(* IEC 61131-3 sources: redes-industriais-mqtt/clp, 4 files *)

(* ---- 1_GVL_MQTT.st ---- *)
(* =========================================================
   GVL_MQTT  -  Global Variable List
   Application > MQTT (pasta) > Add Object > GVL
   ========================================================= *)

VAR_GLOBAL
    (* Estruturas de publicacao e assinatura *)
    Pubs : ARRAY[1..gc_uiMaxPubs] OF MQTT_PUBLISH;
    Subs : ARRAY[1..gc_uiMaxSubs] OF MQTT_SUBSCRIBE;

    (* TOPICOS DE PUBLICACAO - entradas que o CLP envia *)
    PUBLISH_TOPICS : ARRAY[1..gc_uiMaxPubs] OF STRING := [
        'XP340/I_00',
        'XP340/I_01'
    ];

    (* TOPICOS DE ASSINATURA - saidas que o CLP recebe *)
    SUBSCRIBE_TOPICS : ARRAY[1..gc_uiMaxSubs] OF STRING := [
        'XP340/Q_00',
        'XP340/Q_01'
    ];

    (* Status das publicacoes e mensagens recebidas *)
    MQTT_FB_Pub_Status        : ARRAY[1..gc_uiMaxPubs] OF BOOL;
    MQTT_FB_Received_Messages : ARRAY[1..gc_uiMaxSubs] OF MQTT_RECEIVED;

    (* Payloads *)
    PUBS_PAYLOADS : ARRAY[1..gc_uiMaxPubs] OF STRING;
    SUBS_PAYLOADS : ARRAY[1..gc_uiMaxSubs] OF STRING;

    (* Auxiliar - so publica quando o valor muda *)
    PUBS_PAYLOADS_OLD : ARRAY[1..gc_uiMaxPubs] OF STRING;
END_VAR

(* ---- 2_MQTT.st ---- *)
(* =========================================================
   MQTT  -  Program (ST)
   Application > MQTT (pasta) > Add Object > POU
              tipo Program, linguagem Structured Text

   O editor tem DUAS caixas:
   PARTE 1 na de CIMA, PARTE 2 na de BAIXO.
   ========================================================= *)

(* ===== PARTE 1 - CAIXA DE CIMA ===== *)

PROGRAM MQTT
VAR
    MQTT_FB            : MQTT_CLIENT;
    MQTT_FB_Enable     : BOOL := TRUE;
    MQTT_FB_Error      : BOOL;
    MQTT_FB_State      : MQTT_STATES;
    MQTT_FB_Error_Code : MQTT_ERR_CODE;
    i                  : INT;
END_VAR

(* ===== PARTE 2 - CAIXA DE BAIXO ===== *)

(* Conexao com o broker.
   sHostname = IP do PC que roda o docker compose, nao 'mosquitto'.
   O CLP esta fora da rede do Docker e nao resolve esse nome. *)
MQTT_FB.CONNECTION_CONFIG.sHostname     := '192.168.15.10';
MQTT_FB.CONNECTION_CONFIG.uiPort        := 1883;
MQTT_FB.CONNECTION_CONFIG.sClientId     := 'XP340_CLP';
MQTT_FB.CONNECTION_CONFIG.bCleanSession := TRUE;

(* Ponteiros para as variaveis de publicacao e assinatura *)
MQTT_FB.PUBLISH   := Pubs;
MQTT_FB.SUBSCRIBE := Subs;

(* Habilita a funcao MQTT *)
MQTT_FB.ENABLE := MQTT_FB_Enable;

(* Variaveis de erro *)
MQTT_FB_Error      := MQTT_FB.ERROR;
MQTT_FB_State      := MQTT_FB.STATE;
MQTT_FB_Error_Code := MQTT_FB.ERROR_CODE;

(* Status das publicacoes e mensagens recebidas *)
MQTT_FB_Pub_Status        := MQTT_FB.PUBLISH_STATUS;
MQTT_FB_Received_Messages := MQTT_FB.RECEIVED_MESSAGES;

(* Publicacao *)
FOR i := 1 TO TO_INT(gc_uiMaxPubs) DO
    Pubs[i].sPublishTopic        := PUBLISH_TOPICS[i];
    Pubs[i].pbPublishPayload     := ADR(PUBS_PAYLOADS[i]);
    Pubs[i].uiPublishPayloadSize := TO_UINT(LEN(PUBS_PAYLOADS[i]));
    Pubs[i].ePublishMessageQoS   := MQTT_QOS_0;
    Pubs[i].bPublishRetain       := TRUE;

    IF (PUBS_PAYLOADS[i] <> PUBS_PAYLOADS_OLD[i]) THEN
        PUBS_PAYLOADS_OLD[i]   := PUBS_PAYLOADS[i];
        Pubs[i].bEnablePublish := TRUE;
    END_IF

    IF (MQTT_FB_Pub_Status[i]) THEN
        Pubs[i].bEnablePublish := FALSE;
    END_IF
END_FOR

(* Assinatura *)
FOR i := 1 TO TO_INT(gc_uiMaxSubs) DO
    Subs[i].sSubscribeTopic  := SUBSCRIBE_TOPICS[i];
    Subs[i].pbPayloadBuffer  := ADR(SUBS_PAYLOADS[i]);
    Subs[i].uiMaxPayloadSize := SIZEOF(SUBS_PAYLOADS[i]);
    Subs[i].eSubscribeQoS    := MQTT_QOS_0;
END_FOR

(* Reconexao em caso de falha *)
IF MQTT_FB_Error THEN
    MQTT_FB_Enable := PULSE_5S;
ELSE
    MQTT_FB_Enable := TRUE;
END_IF

(* Chamada do bloco *)
MQTT_FB();

(* ---- 3_ESPELHAMENTO_ENTRADAS_MQTT.st ---- *)
(* =========================================================
   ESPELHAMENTO_ENTRADAS_MQTT  -  Program (ST)
   Le as entradas fisicas e monta os payloads de publicacao.
   Payload ON/OFF para casar com o dashboard.
   ========================================================= *)

(* ===== PARTE 1 - CAIXA DE CIMA ===== *)

PROGRAM ESPELHAMENTO_ENTRADAS_MQTT
VAR
END_VAR

(* ===== PARTE 2 - CAIXA DE BAIXO ===== *)

IF I00 THEN
    PUBS_PAYLOADS[1] := 'ON';
ELSE
    PUBS_PAYLOADS[1] := 'OFF';
END_IF

IF I01 THEN
    PUBS_PAYLOADS[2] := 'ON';
ELSE
    PUBS_PAYLOADS[2] := 'OFF';
END_IF

(* ---- 4_ESPELHAMENTO_SAIDAS_MQTT.st ---- *)
(* =========================================================
   ESPELHAMENTO_SAIDAS_MQTT  -  Program (ST)
   Converte os payloads recebidos e aciona as saidas fisicas.
   ========================================================= *)

(* ===== PARTE 1 - CAIXA DE CIMA ===== *)

PROGRAM ESPELHAMENTO_SAIDAS_MQTT
VAR
END_VAR

(* ===== PARTE 2 - CAIXA DE BAIXO ===== *)

Q00 := (SUBS_PAYLOADS[1] = 'ON');
Q01 := (SUBS_PAYLOADS[2] = 'ON');
